(* Schneider Machine Expert - Basic project Proyecto_PLC_M221_Alex, file version 3.0.0.0 *)
(* CompanyInformations: Name=Alex, Country=España *)
(* ProjectInformations: Name=Proyecto1_PLC_M221_Alex, Description=Proyecto 1 Schneider Electric con M221.

Se ha a realizado el control de una maqueta Fischertechnik, la cual es una
línea de fabricación con dos máquinas herramienta, cinco cintas y dos selectores.

Se han realizado:
	- Diagrama de cableado de la maqueta.
	‐ Red de Petri
	‐ Implementación mediante Grafcet (las secciones LD)
	- Implementación de diferentes modos de la guía Gemma.
	‐ Implementar el panel de control de la máquina en un terminal de explotación. *)
(* UserInformations: LastName=Aquino Sala, FirstName=Alex, Email=aaleexsaalaa@gmail.com, Country=España *)

HARDWARE
  Cpu 0: TM221CE24R
  EthernetConfiguration: NetworkName=M221, IpAllocationMode=FixedAddress, IpAddress=10.7.1.158, SubnetMask=255.255.255.0
  SerialLineConfiguration: Baud=Baud19200, Parity=ParityEven, DataBits=DataBits8, StopBits=StopBits1, PhysicalMedium=PhysicalMediumRs485, TransmissionMode=TransmissionModeModbusRtu, SlaveId=1, Addressing=SlaveAddressing
  MastTask: UsePeriodScanMode=false, PeriodScan=100
  FastTask: Period=255
  CpuBehavior: StartingMode=StartAsPreviousState, AutoSaveRamOnEeprom=true, WatchdogPeriod=250

SYMBOLS  (address, symbol, comment, settings)
  %M100     AUTO  "Bit para poner el modo automatico"
  %M101     G_QCINTA1  "Bit para el control del modo manual"
  %M102     G_QCINTA2  "Bit para el control del modo manual"
  %M103     G_QCINTA3  "Bit para el control del modo manual"
  %M104     G_QCINTA4  "Bit para el control del modo manual"
  %M105     G_QMAC1  "Bit para el control del modo manual"
  %M106     G_QMAC2  "Bit para el control del modo manual"
  %M107     G_QSEL1AVANZA  "Bit para el control del modo manual"
  %M108     G_QSEL1RETRO  "Bit para el control del modo manual"
  %M109     G_QSEL2AVANZA  "Bit para el control del modo manual"
  %M110     G_QSEL2RETRO  "Bit para el control del modo manual"
  %M111     MARCHA
  %M112     EMERGENCIA  "Bit emergencia"
  %M113     REARME  "Bit de rearme"
  %M200     ESTOY_EMERG  "Bit que indica que esta en emergencia"
  %M201     ESTOY_MANUAL  "Bit para indicar cuando estamos en manual"
  %M202     ESTOY_AUTO  "Bit que indica cuando esta en modo automatico"
  %M300     PROBLEMAC1  "Problema en cinta 1"
  %M301     PROBLEMAC2  "Problema en cinta 2"
  %M302     PROBLEMAC3  "Problema en cinta 3"
  %M303     PROBLEMAC4  "Problema en cinta 4"
  %M304     PROBLEMA_MQ1  "Problema en maquina 1"
  %M305     PROBLEMA_MQ2  "Problema en maquina 2"
  %S9       SB_FALLBACKOUTPUT  "Establézcalo en 1 para aplicar retornos en salidas digitales y analógicas"
  %S23      SB_FREEZEGRAFCET  "Cuando es 1, valida el posicionamiento previo del GRAFCET. Si se mantiene este bit en 1, se inmoviliza el GRAFCET (se inmoviliza el gráfico)"
  %X2         "C1 avanza"
  %X3         "Espera C1"
  %X4         "R1 avanza"
  %X5         "C2 avanza"
  %X6         "Maquina 1 trabaja"
  %X8         "Maquina 2 trabaja"
  %X9         "Maquina 2 trabaja"
  %X10        "Espera M2"
  %X11        "C3 avanza"
  %X12        "R2 avanza"
  %X13        "C4 avanza"
  %X15        "R1 retrocede"
  %X16        "Espera"
  %X17        "R2 avanza"
  %X18        "Espera"
  %X19        "C1 avanza"
  %X20        "Epera R1"
  %X21        "Espera R2"
  %X23        "F4"
  %X24        "A6"
  %X25        "F1"
  %TM0        "Temporizador para los segundos de la maquina 1"  [Preset=5, Base=OneSecond]
  %TM1        "Temporizador para los segundos de la maquina 2"  [Preset=10, Base=OneSecond]
  %TM2        "Temporizador para que llegue la pieza al final de la cinta"  [Preset=7, Base=OneHundredMilliSeconds]
  %TM3        "Temporizador para que llegue la pieza al final de la cinta"  [Preset=2, Base=OneSecond]
  %TM4        "Temporizador que controla los problemas"  [Preset=7, Base=OneSecond]
  %TM5        "Temporizador que controla los problemas"  [Preset=7, Base=OneSecond]
  %TM6        "Temporizador que controla los problemas"  [Preset=7, Base=OneSecond]
  %TM7        "Temporizador que controla los problemas"  [Preset=7, Base=OneSecond]
  %TM8        "Temporizador que controla los problemas"  [Preset=7, Base=OneSecond]
  %TM9        "Temporizador que controla los problemas"  [Preset=12, Base=OneSecond]
  %I0.0     ISEL1FIN  "selector 1"
  %I0.1     ISENSORC1  "sensor 1"
  %I0.2     ISENSORCARGA
  %I0.3     ISENSORMAQ1  "sensor maquina"
  %I0.4     ISENSORMAQ2  "sensor maquina 2"
  %I0.5     ISEL1INI  "Selecrtor 1"
  %I0.6     ISENSORC4  "sensor 4"
  %I0.7     ISEL2FIN  "selecotr 2 fin"
  %I0.8     ISEL2INI  "Selector 2 ini"
  %Q0.0     QSEL1AVANZA  "Bit para mover el selector"
  %Q0.1     QMAQ1  "Bit para activar la maquina 1"
  %Q0.2     QCINTA3  "Bit para mover la cinta 3"
  %Q0.3     QSEL1RETRO  "Bit para mover el selector"
  %Q0.4     QSEL2AVANZA  "Bit para mover el selector"
  %Q0.5     QCINTA1  "Bit para mover la cinta 1"
  %Q0.6     QCINTA2  "Bit para mover la cinta 2"
  %Q0.7     QSEL2RETRO  "Bit para mover el selector"
  %Q0.8     QMAQ2  "Bit para activar la maquina"
  %Q0.9     QCINTA4  "Bit para mover la cinta 4"

GRAFCET GEMMA
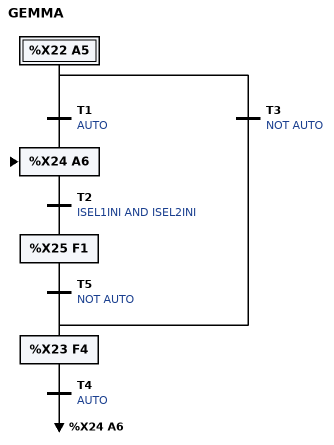
  INITIAL_STEP %X22  (* A5 *)
  STEP %X23  (* F4 *)
  STEP %X24  (* A6 *)
  STEP %X25  (* F1 *)
  TRANSITION T1 FROM %X22 TO %X24 := AUTO;
  TRANSITION T2 FROM %X24 TO %X25 := ISEL1INI AND ISEL2INI;
  TRANSITION T3 FROM %X22 TO %X23 := NOT AUTO;
  TRANSITION T4 FROM %X23 TO %X24 := AUTO;
  TRANSITION T5 FROM %X25 TO %X23 := NOT AUTO;

GRAFCET GRAFET
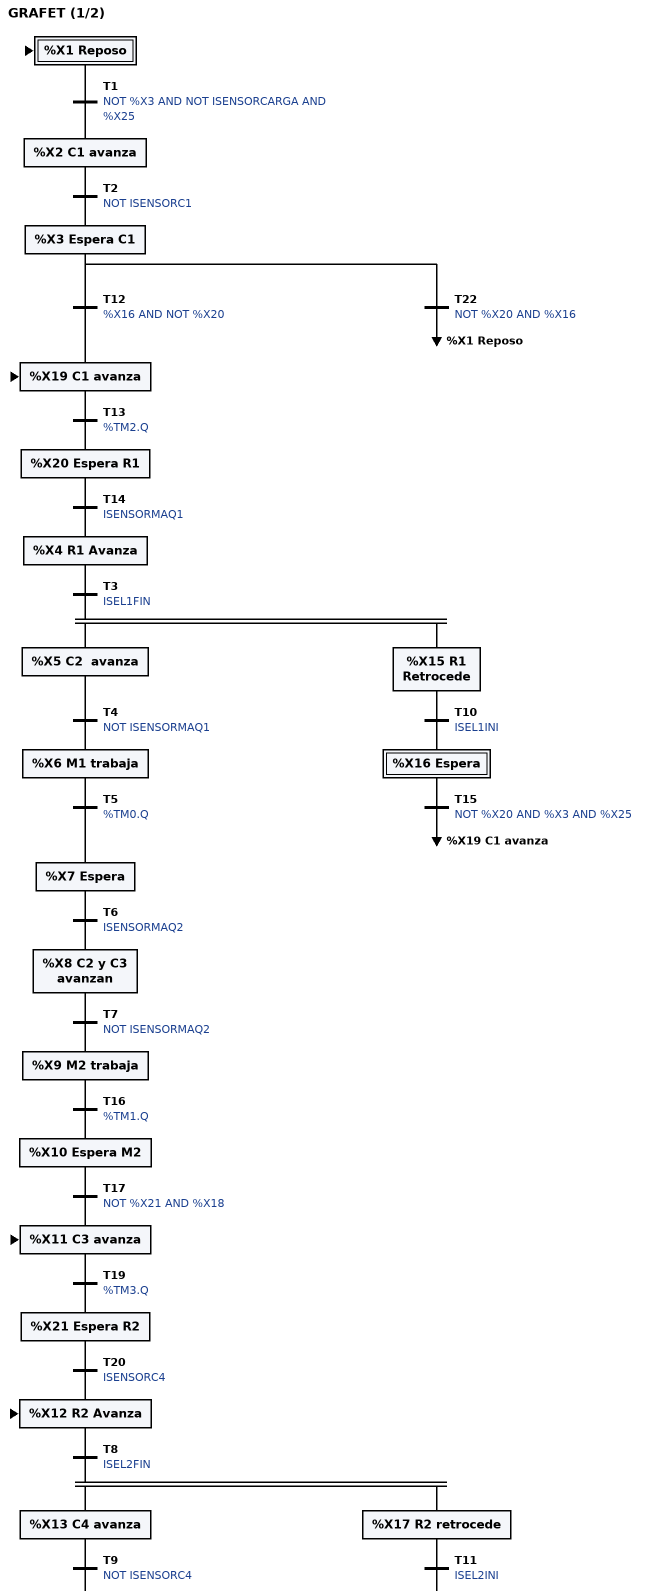
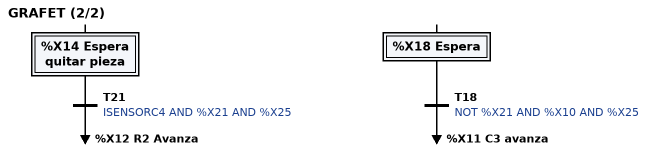
  INITIAL_STEP %X1  (* Reposo *)
  STEP %X2  (* C1 avanza *)
  STEP %X3  (* Espera C1 *)
  STEP %X4  (* R1 Avanza *)
  STEP %X5  (* C2  avanza *)
  STEP %X6  (* M1 trabaja *)
  STEP %X7  (* Espera *)
  STEP %X8  (* C2 y C3 avanzan *)
  STEP %X9  (* M2 trabaja *)
  STEP %X10  (* Espera M2 *)
  STEP %X11  (* C3 avanza *)
  STEP %X12  (* R2 Avanza *)
  STEP %X13  (* C4 avanza *)
  INITIAL_STEP %X14  (* Espera quitar pieza *)
  STEP %X15  (* R1 Retrocede *)
  INITIAL_STEP %X16  (* Espera  *)
  STEP %X17  (* R2 retrocede *)
  INITIAL_STEP %X18  (* Espera *)
  STEP %X19  (* C1 avanza *)
  STEP %X20  (* Espera R1 *)
  STEP %X21  (* Espera R2 *)
  TRANSITION T1 FROM %X1 TO %X2 := NOT %X3 AND NOT ISENSORCARGA AND %X25;
  TRANSITION T2 FROM %X2 TO %X3 := NOT ISENSORC1;
  TRANSITION T3 FROM %X4 TO %X5, %X15 := ISEL1FIN;
  TRANSITION T4 FROM %X5 TO %X6 := NOT ISENSORMAQ1;
  TRANSITION T5 FROM %X6 TO %X7 := %TM0.Q;
  TRANSITION T6 FROM %X7 TO %X8 := ISENSORMAQ2;
  TRANSITION T7 FROM %X8 TO %X9 := NOT ISENSORMAQ2;
  TRANSITION T8 FROM %X12 TO %X13, %X17 := ISEL2FIN;
  TRANSITION T9 FROM %X13 TO %X14 := NOT ISENSORC4;
  TRANSITION T10 FROM %X15 TO %X16 := ISEL1INI;
  TRANSITION T11 FROM %X17 TO %X18 := ISEL2INI;
  TRANSITION T12 FROM %X3 TO %X19 := %X16 AND NOT %X20;
  TRANSITION T13 FROM %X19 TO %X20 := %TM2.Q;
  TRANSITION T14 FROM %X20 TO %X4 := ISENSORMAQ1;
  TRANSITION T15 FROM %X16 TO %X19 := NOT %X20 AND %X3 AND %X25;
  TRANSITION T16 FROM %X9 TO %X10 := %TM1.Q;
  TRANSITION T17 FROM %X10 TO %X11 := NOT %X21 AND %X18;
  TRANSITION T18 FROM %X18 TO %X11 := NOT %X21 AND %X10 AND %X25;
  TRANSITION T19 FROM %X11 TO %X21 := %TM3.Q;
  TRANSITION T20 FROM %X21 TO %X12 := ISENSORC4;
  TRANSITION T21 FROM %X14 TO %X12 := ISENSORC4 AND %X21 AND %X25;
  TRANSITION T22 FROM %X3 TO %X1 := NOT %X20 AND %X16;

TRANSITION T1 (%X22 -> %X24) 
  (* SectionNumber=0 *)

// Rung 0: AUTO
  LD %M100                (* AUTO *)
  ENDT
  // as ST:
  //   TRANSITION := AUTO;

TRANSITION T2 (%X24 -> %X25) 
  (* SectionNumber=0 *)

// Rung 1: Tr2
  LD %I0.5                (* ISEL1INI *)
  AND %I0.8               (* ISEL2INI *)
  ENDT
  // as ST:
  //   TRANSITION := ISEL1INI AND ISEL2INI;

TRANSITION T3 (%X22 -> %X23) 
  (* SectionNumber=0 *)

// Rung 2: MANUAL
  LDN %M100               (* AUTO *)
  ENDT
  // as ST:
  //   TRANSITION := NOT AUTO;

TRANSITION T4 (%X23 -> %X24) 
  (* SectionNumber=0 *)

// Rung 3: AUTO
  LD %M100                (* AUTO *)
  ENDT
  // as ST:
  //   TRANSITION := AUTO;

TRANSITION T5 (%X25 -> %X23) 
  (* SectionNumber=0 *)

// Rung 4: MANUAL
  LDN %M100               (* AUTO *)
  ENDT
  // as ST:
  //   TRANSITION := NOT AUTO;

TRANSITION T1 (%X1 -> %X2) 
  (* SectionNumber=0 *)

// Rung 5: Tr1
  LDN %X3
  ANDN %I0.2              (* ISENSORCARGA *)
  AND %X25
  ENDT
  // as ST:
  //   TRANSITION := NOT %X3 AND NOT ISENSORCARGA AND %X25;

TRANSITION T2 (%X2 -> %X3) 
  (* SectionNumber=0 *)

// Rung 6: Tr2
  LDN %I0.1               (* ISENSORC1 *)
  ENDT
  // as ST:
  //   TRANSITION := NOT ISENSORC1;

TRANSITION T3 (%X4 -> %X5, %X15) 
  (* SectionNumber=0 *)

// Rung 7: Tr4
  LD %I0.0                (* ISEL1FIN *)
  ENDT
  // as ST:
  //   TRANSITION := ISEL1FIN;

TRANSITION T4 (%X5 -> %X6) 
  (* SectionNumber=0 *)

// Rung 8: Tr5
  LDN %I0.3               (* ISENSORMAQ1 *)
  ENDT
  // as ST:
  //   TRANSITION := NOT ISENSORMAQ1;

TRANSITION T5 (%X6 -> %X7) 
  (* SectionNumber=0 *)

// Rung 9: Temp
  LD %TM0.Q
  ENDT
  // as ST:
  //   TRANSITION := %TM0.Q;

TRANSITION T6 (%X7 -> %X8) 
  (* SectionNumber=0 *)

// Rung 10: Tr7
  LD %I0.4                (* ISENSORMAQ2 *)
  ENDT
  // as ST:
  //   TRANSITION := ISENSORMAQ2;

TRANSITION T7 (%X8 -> %X9) 
  (* SectionNumber=0 *)

// Rung 11: Tr8
  LDN %I0.4               (* ISENSORMAQ2 *)
  ENDT
  // as ST:
  //   TRANSITION := NOT ISENSORMAQ2;

TRANSITION T8 (%X12 -> %X13, %X17) 
  (* SectionNumber=0 *)

// Rung 12: Tr12
  LD %I0.7                (* ISEL2FIN *)
  ENDT
  // as ST:
  //   TRANSITION := ISEL2FIN;

TRANSITION T9 (%X13 -> %X14) 
  (* SectionNumber=0 *)

// Rung 13: Tr13
  LDN %I0.6               (* ISENSORC4 *)
  ENDT
  // as ST:
  //   TRANSITION := NOT ISENSORC4;

TRANSITION T10 (%X15 -> %X16) 
  (* SectionNumber=0 *)

// Rung 14: Tr14
  LD %I0.5                (* ISEL1INI *)
  ENDT
  // as ST:
  //   TRANSITION := ISEL1INI;

TRANSITION T11 (%X17 -> %X18) 
  (* SectionNumber=0 *)

// Rung 15: Tr16
  LD %I0.8                (* ISEL2INI *)
  ENDT
  // as ST:
  //   TRANSITION := ISEL2INI;

TRANSITION T12 (%X3 -> %X19) 
  (* SectionNumber=0 *)

// Rung 16: Tr3
  LD %X16
  ANDN %X20
  ENDT
  // as ST:
  //   TRANSITION := %X16 AND NOT %X20;

TRANSITION T13 (%X19 -> %X20) 
  (* SectionNumber=0 *)

// Rung 17: Temp
  LD %TM2.Q
  ENDT
  // as ST:
  //   TRANSITION := %TM2.Q;

TRANSITION T14 (%X20 -> %X4) 
  (* SectionNumber=0 *)

// Rung 18: Tr19
  LD %I0.3                (* ISENSORMAQ1 *)
  ENDT
  // as ST:
  //   TRANSITION := ISENSORMAQ1;

TRANSITION T15 (%X16 -> %X19) 
  (* SectionNumber=0 *)

// Rung 19: Tr20
  LDN %X20
  AND %X3
  AND %X25
  ENDT
  // as ST:
  //   TRANSITION := NOT %X20 AND %X3 AND %X25;

TRANSITION T16 (%X9 -> %X10) 
  (* SectionNumber=0 *)

// Rung 20: Temp
  LD %TM1.Q
  ENDT
  // as ST:
  //   TRANSITION := %TM1.Q;

TRANSITION T17 (%X10 -> %X11) 
  (* SectionNumber=0 *)

// Rung 21: Tr13
  LDN %X21
  AND %X18
  ENDT
  // as ST:
  //   TRANSITION := NOT %X21 AND %X18;

TRANSITION T18 (%X18 -> %X11) 
  (* SectionNumber=0 *)

// Rung 22: Tr13
  LDN %X21
  AND %X10
  AND %X25
  ENDT
  // as ST:
  //   TRANSITION := NOT %X21 AND %X10 AND %X25;

TRANSITION T19 (%X11 -> %X21) 
  (* SectionNumber=0 *)

// Rung 23: Temp
  LD %TM3.Q
  ENDT
  // as ST:
  //   TRANSITION := %TM3.Q;

TRANSITION T20 (%X21 -> %X12) 
  (* SectionNumber=0 *)

// Rung 24: Tr14
  LD %I0.6                (* ISENSORC4 *)
  ENDT
  // as ST:
  //   TRANSITION := ISENSORC4;

TRANSITION T21 (%X14 -> %X12) 
  (* SectionNumber=0 *)

// Rung 25: Tr21
  LD %I0.6                (* ISENSORC4 *)
  AND %X21
  AND %X25
  ENDT
  // as ST:
  //   TRANSITION := ISENSORC4 AND %X21 AND %X25;

TRANSITION T22 (%X3 -> %X1) 
  (* SectionNumber=0 *)

// Rung 26: Tr22
  LDN %X20
  AND %X16
  ENDT
  // as ST:
  //   TRANSITION := NOT %X20 AND %X16;

POU SALIDAS  (* Lineas para controlar las salidas de nuestro sistema *)
  (* SectionNumber=27 *)

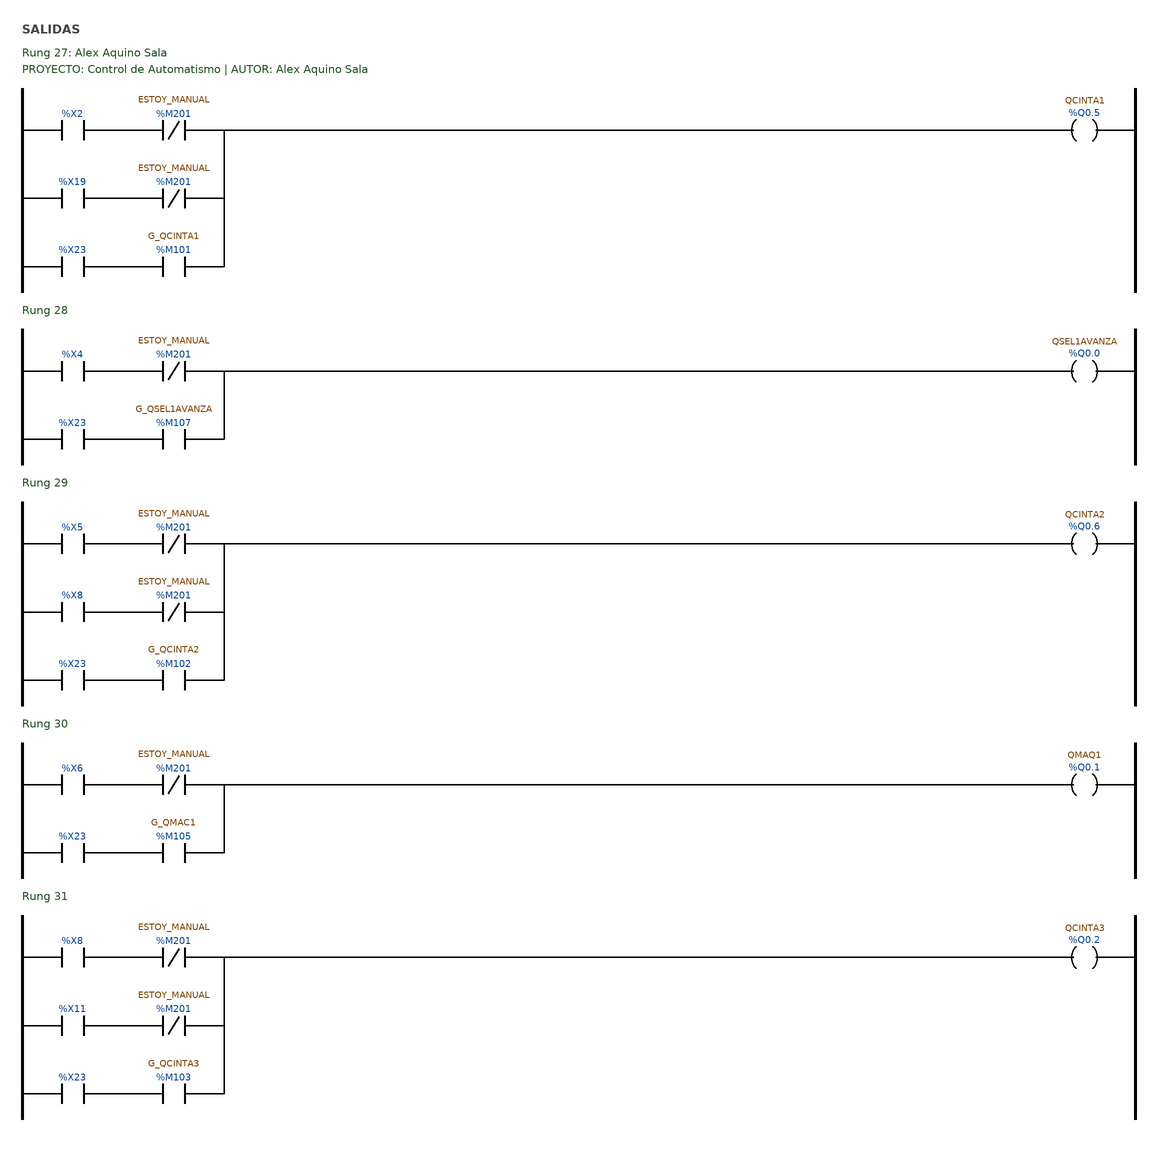

// Rung 27: Alex Aquino Sala
// PROYECTO: Control de Automatismo | AUTOR: Alex Aquino Sala
  LD %X2
  ANDN %M201              (* ESTOY_MANUAL *)
  OR( %X19
  ANDN %M201              (* ESTOY_MANUAL *)
  )
  OR( %X23
  AND %M101               (* G_QCINTA1 *)
  )
  ST %Q0.5                (* QCINTA1 *)
  // as ST:
  //   QCINTA1 := %X2 AND NOT ESTOY_MANUAL OR %X19 AND NOT ESTOY_MANUAL OR %X23 AND G_QCINTA1;

// Rung 28
  LD %X4
  ANDN %M201              (* ESTOY_MANUAL *)
  OR( %X23
  AND %M107               (* G_QSEL1AVANZA *)
  )
  ST %Q0.0                (* QSEL1AVANZA *)
  // as ST:
  //   QSEL1AVANZA := %X4 AND NOT ESTOY_MANUAL OR %X23 AND G_QSEL1AVANZA;

// Rung 29
  LD %X5
  ANDN %M201              (* ESTOY_MANUAL *)
  OR( %X8
  ANDN %M201              (* ESTOY_MANUAL *)
  )
  OR( %X23
  AND %M102               (* G_QCINTA2 *)
  )
  ST %Q0.6                (* QCINTA2 *)
  // as ST:
  //   QCINTA2 := %X5 AND NOT ESTOY_MANUAL OR %X8 AND NOT ESTOY_MANUAL OR %X23 AND G_QCINTA2;

// Rung 30
  LD %X6
  ANDN %M201              (* ESTOY_MANUAL *)
  OR( %X23
  AND %M105               (* G_QMAC1 *)
  )
  ST %Q0.1                (* QMAQ1 *)
  // as ST:
  //   QMAQ1 := %X6 AND NOT ESTOY_MANUAL OR %X23 AND G_QMAC1;

// Rung 31
  LD %X8
  ANDN %M201              (* ESTOY_MANUAL *)
  OR( %X11
  ANDN %M201              (* ESTOY_MANUAL *)
  )
  OR( %X23
  AND %M103               (* G_QCINTA3 *)
  )
  ST %Q0.2                (* QCINTA3 *)
  // as ST:
  //   QCINTA3 := %X8 AND NOT ESTOY_MANUAL OR %X11 AND NOT ESTOY_MANUAL OR %X23 AND G_QCINTA3;

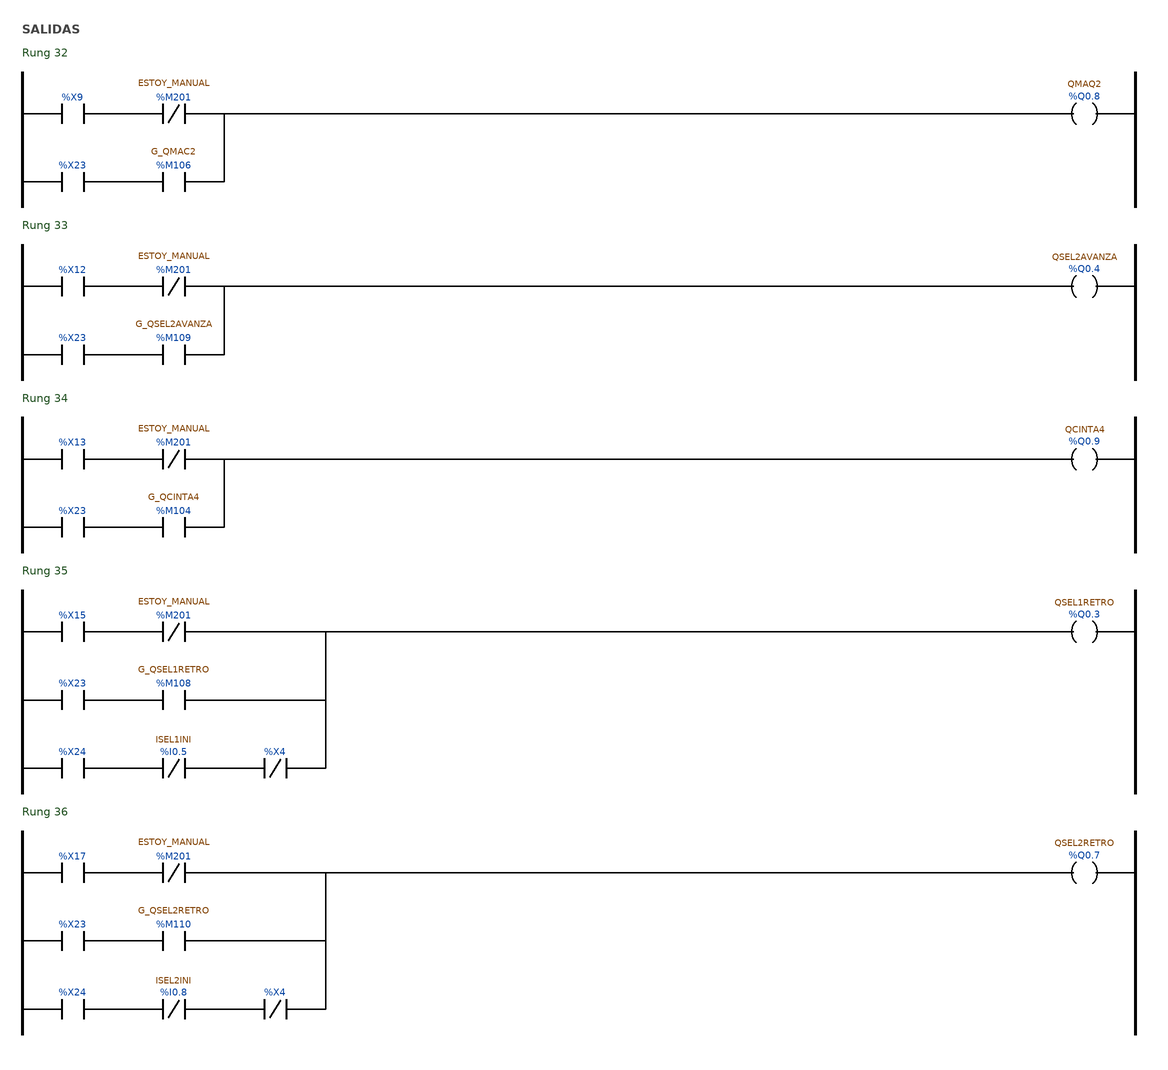

// Rung 32
  LD %X9
  ANDN %M201              (* ESTOY_MANUAL *)
  OR( %X23
  AND %M106               (* G_QMAC2 *)
  )
  ST %Q0.8                (* QMAQ2 *)
  // as ST:
  //   QMAQ2 := %X9 AND NOT ESTOY_MANUAL OR %X23 AND G_QMAC2;

// Rung 33
  LD %X12
  ANDN %M201              (* ESTOY_MANUAL *)
  OR( %X23
  AND %M109               (* G_QSEL2AVANZA *)
  )
  ST %Q0.4                (* QSEL2AVANZA *)
  // as ST:
  //   QSEL2AVANZA := %X12 AND NOT ESTOY_MANUAL OR %X23 AND G_QSEL2AVANZA;

// Rung 34
  LD %X13
  ANDN %M201              (* ESTOY_MANUAL *)
  OR( %X23
  AND %M104               (* G_QCINTA4 *)
  )
  ST %Q0.9                (* QCINTA4 *)
  // as ST:
  //   QCINTA4 := %X13 AND NOT ESTOY_MANUAL OR %X23 AND G_QCINTA4;

// Rung 35
  LD %X15
  ANDN %M201              (* ESTOY_MANUAL *)
  OR( %X23
  AND %M108               (* G_QSEL1RETRO *)
  )
  OR( %X24
  ANDN %I0.5              (* ISEL1INI *)
  ANDN %X4
  )
  ST %Q0.3                (* QSEL1RETRO *)
  // as ST:
  //   QSEL1RETRO := %X15 AND NOT ESTOY_MANUAL OR %X23 AND G_QSEL1RETRO OR %X24 AND NOT ISEL1INI AND NOT %X4;

// Rung 36
  LD %X17
  ANDN %M201              (* ESTOY_MANUAL *)
  OR( %X23
  AND %M110               (* G_QSEL2RETRO *)
  )
  OR( %X24
  ANDN %I0.8              (* ISEL2INI *)
  ANDN %X4
  )
  ST %Q0.7                (* QSEL2RETRO *)
  // as ST:
  //   QSEL2RETRO := %X17 AND NOT ESTOY_MANUAL OR %X23 AND G_QSEL2RETRO OR %X24 AND NOT ISEL2INI AND NOT %X4;

POU MODOS  (* Lineas para comunicar con el HMI *)
  (* SectionNumber=28 *)

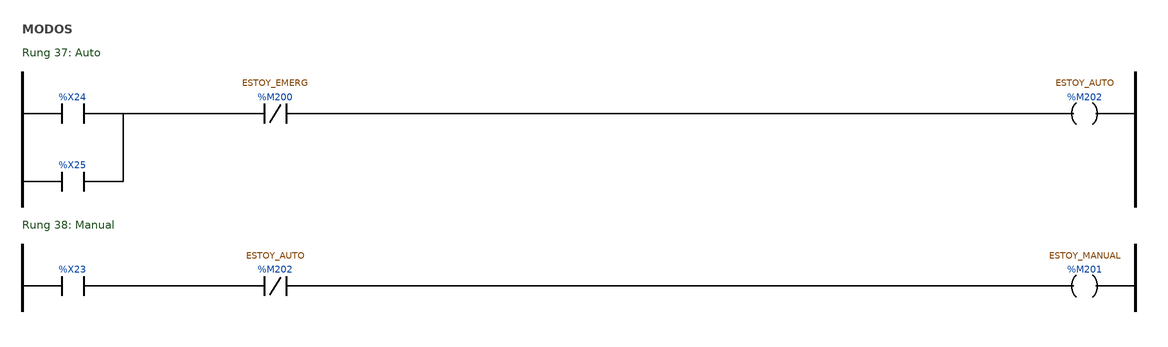

// Rung 37: Auto
  LD %X24
  OR %X25
  ANDN %M200              (* ESTOY_EMERG *)
  ST %M202                (* ESTOY_AUTO *)
  // as ST:
  //   ESTOY_AUTO := (%X24 OR %X25) AND NOT ESTOY_EMERG;

// Rung 38: Manual
  LD %X23
  ANDN %M202              (* ESTOY_AUTO *)
  ST %M201                (* ESTOY_MANUAL *)
  // as ST:
  //   ESTOY_MANUAL := %X23 AND NOT ESTOY_AUTO;

POU TEMPORIZADORES
  (* SectionNumber=29 *)

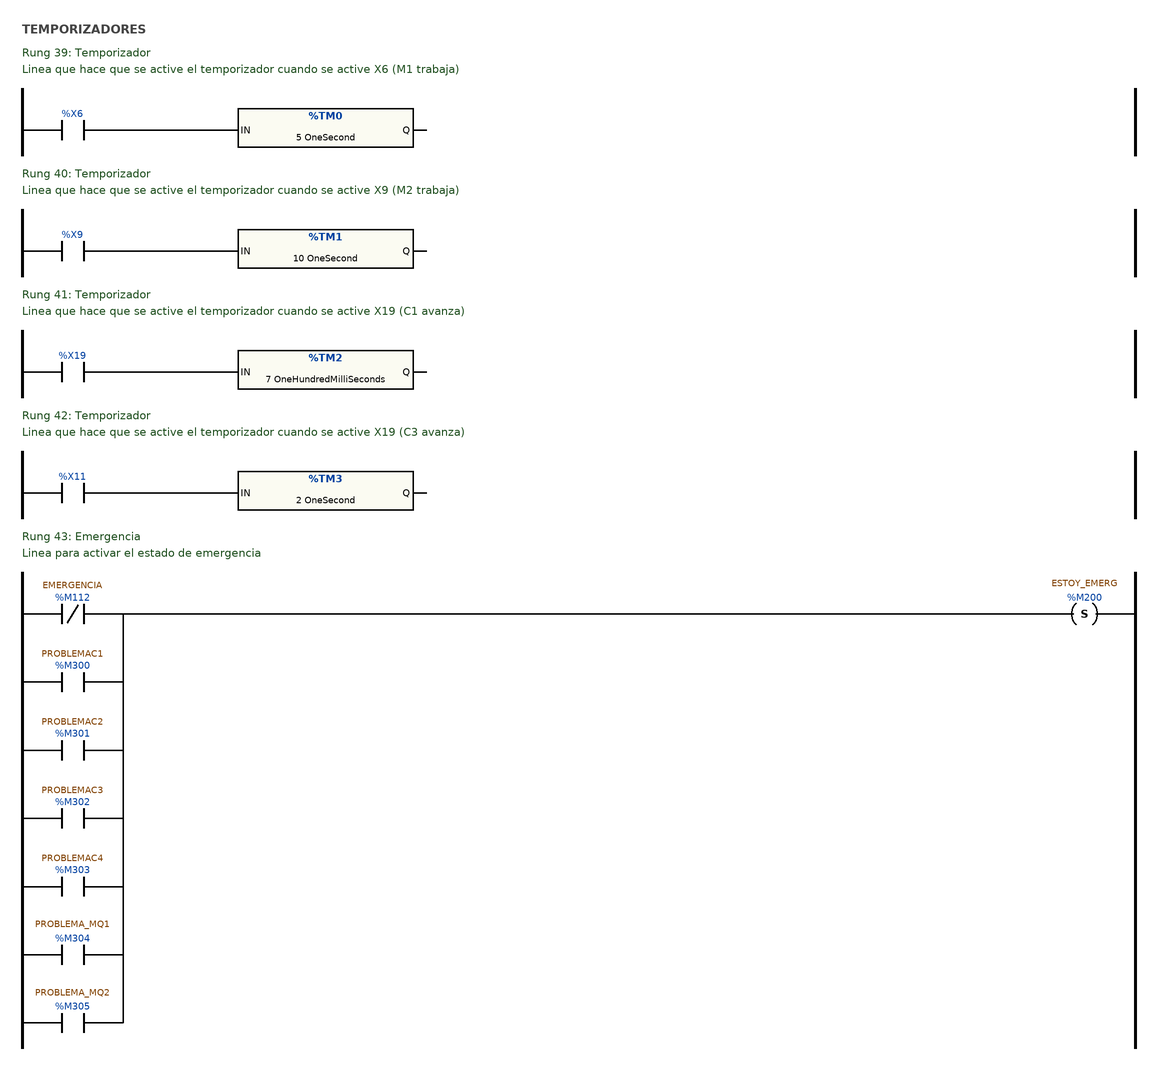

// Rung 39: Temporizador
// Linea que hace que se active el temporizador cuando se active X6 (M1 trabaja)
  BLK %TM0
  LD %X6
  IN
  END_BLK
  // as ST:
  //   %TM0(IN := %X6);

// Rung 40: Temporizador
// Linea que hace que se active el temporizador cuando se active X9 (M2 trabaja)
  BLK %TM1
  LD %X9
  IN
  END_BLK
  // as ST:
  //   %TM1(IN := %X9);

// Rung 41: Temporizador
// Linea que hace que se active el temporizador cuando se active X19 (C1 avanza)
  BLK %TM2
  LD %X19
  IN
  END_BLK
  // as ST:
  //   %TM2(IN := %X19);

// Rung 42: Temporizador
// Linea que hace que se active el temporizador cuando se active X19 (C3 avanza)
  BLK %TM3
  LD %X11
  IN
  END_BLK
  // as ST:
  //   %TM3(IN := %X11);

// Rung 43: Emergencia
// Linea para activar el estado de emergencia
  LDN %M112               (* EMERGENCIA *)
  OR %M300                (* PROBLEMAC1 *)
  OR %M301                (* PROBLEMAC2 *)
  OR %M302                (* PROBLEMAC3 *)
  OR %M303                (* PROBLEMAC4 *)
  OR %M304                (* PROBLEMA_MQ1 *)
  OR %M305                (* PROBLEMA_MQ2 *)
  S %M200                 (* ESTOY_EMERG *)
  // as ST:
  //   IF NOT EMERGENCIA OR PROBLEMAC1 OR PROBLEMAC2 OR PROBLEMAC3 OR PROBLEMAC4 OR PROBLEMA_MQ1 OR PROBLEMA_MQ2 THEN ESTOY_EMERG := TRUE; END_IF;

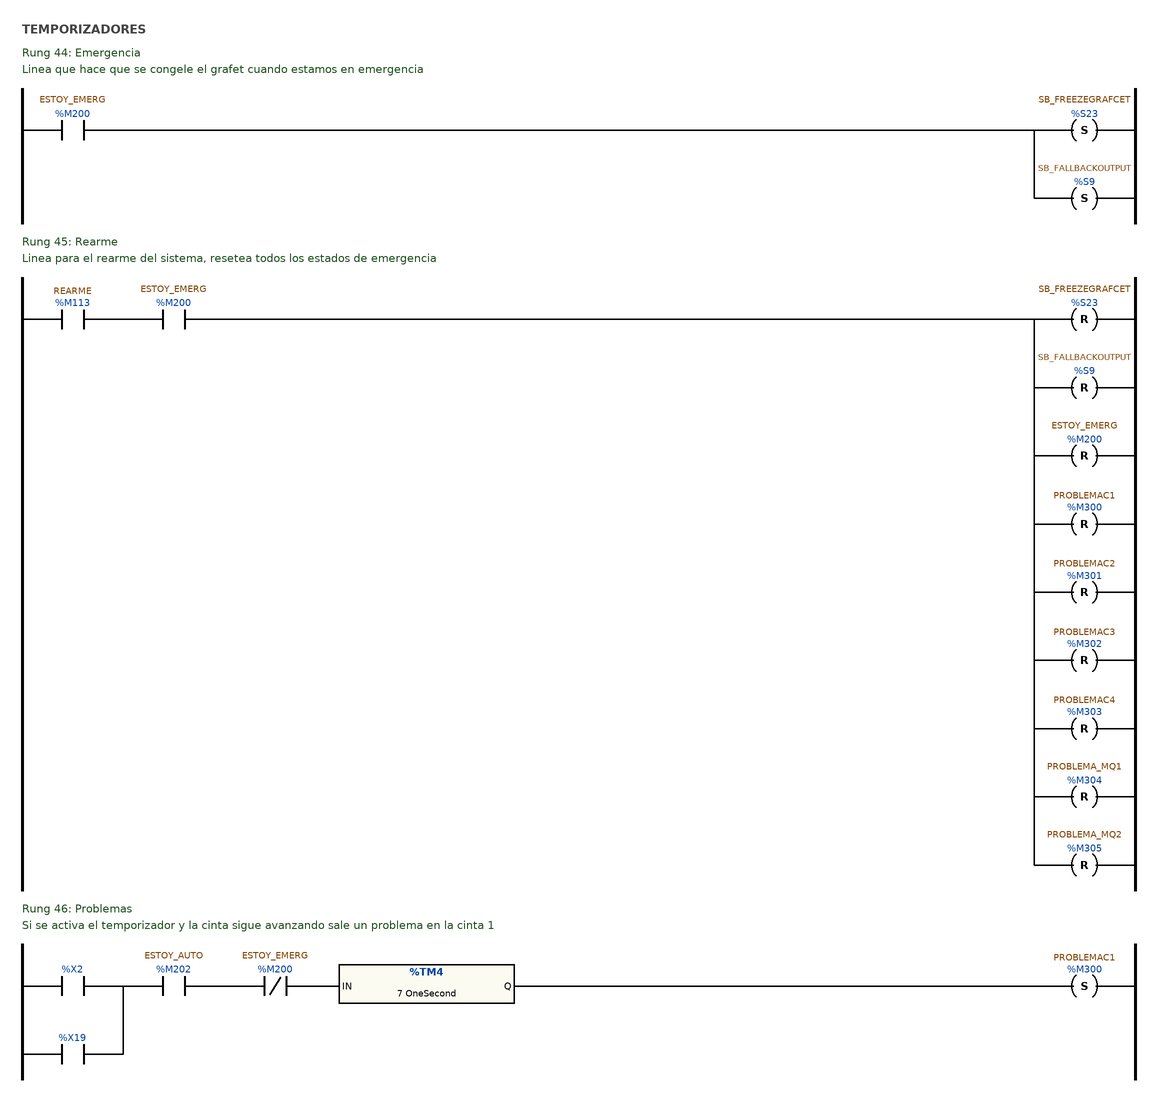

// Rung 44: Emergencia
// Linea que hace que se congele el grafet cuando estamos en emergencia
  LD %M200                (* ESTOY_EMERG *)
  S %S23                  (* SB_FREEZEGRAFCET *)
  S %S9                   (* SB_FALLBACKOUTPUT *)
  // as ST:
  //   IF ESTOY_EMERG THEN SB_FREEZEGRAFCET := TRUE; END_IF;
  //   IF ESTOY_EMERG THEN SB_FALLBACKOUTPUT := TRUE; END_IF;

// Rung 45: Rearme
// Linea para el rearme del sistema, resetea todos los estados de emergencia
  LD %M113                (* REARME *)
  AND %M200               (* ESTOY_EMERG *)
  R %S23                  (* SB_FREEZEGRAFCET *)
  R %S9                   (* SB_FALLBACKOUTPUT *)
  R %M200                 (* ESTOY_EMERG *)
  R %M300                 (* PROBLEMAC1 *)
  R %M301                 (* PROBLEMAC2 *)
  R %M302                 (* PROBLEMAC3 *)
  R %M303                 (* PROBLEMAC4 *)
  R %M304                 (* PROBLEMA_MQ1 *)
  R %M305                 (* PROBLEMA_MQ2 *)
  // as ST:
  //   IF REARME AND ESTOY_EMERG THEN SB_FREEZEGRAFCET := FALSE; END_IF;
  //   IF REARME AND ESTOY_EMERG THEN SB_FALLBACKOUTPUT := FALSE; END_IF;
  //   _t1 := REARME AND ESTOY_EMERG;
  //   IF _t1 THEN ESTOY_EMERG := FALSE; END_IF;
  //   IF _t1 THEN PROBLEMAC1 := FALSE; END_IF;
  //   IF _t1 THEN PROBLEMAC2 := FALSE; END_IF;
  //   IF _t1 THEN PROBLEMAC3 := FALSE; END_IF;
  //   IF _t1 THEN PROBLEMAC4 := FALSE; END_IF;
  //   IF _t1 THEN PROBLEMA_MQ1 := FALSE; END_IF;
  //   IF _t1 THEN PROBLEMA_MQ2 := FALSE; END_IF;

// Rung 46: Problemas
// Si se activa el temporizador y la cinta sigue avanzando sale un problema en la cinta 1
  BLK %TM4
  LD %X2
  OR %X19
  AND %M202               (* ESTOY_AUTO *)
  ANDN %M200              (* ESTOY_EMERG *)
  IN
  OUT_BLK
  LD Q
  S %M300                 (* PROBLEMAC1 *)
  END_BLK
  // as ST:
  //   %TM4(IN := (%X2 OR %X19) AND ESTOY_AUTO AND NOT ESTOY_EMERG);
  //   IF %TM4.Q THEN PROBLEMAC1 := TRUE; END_IF;

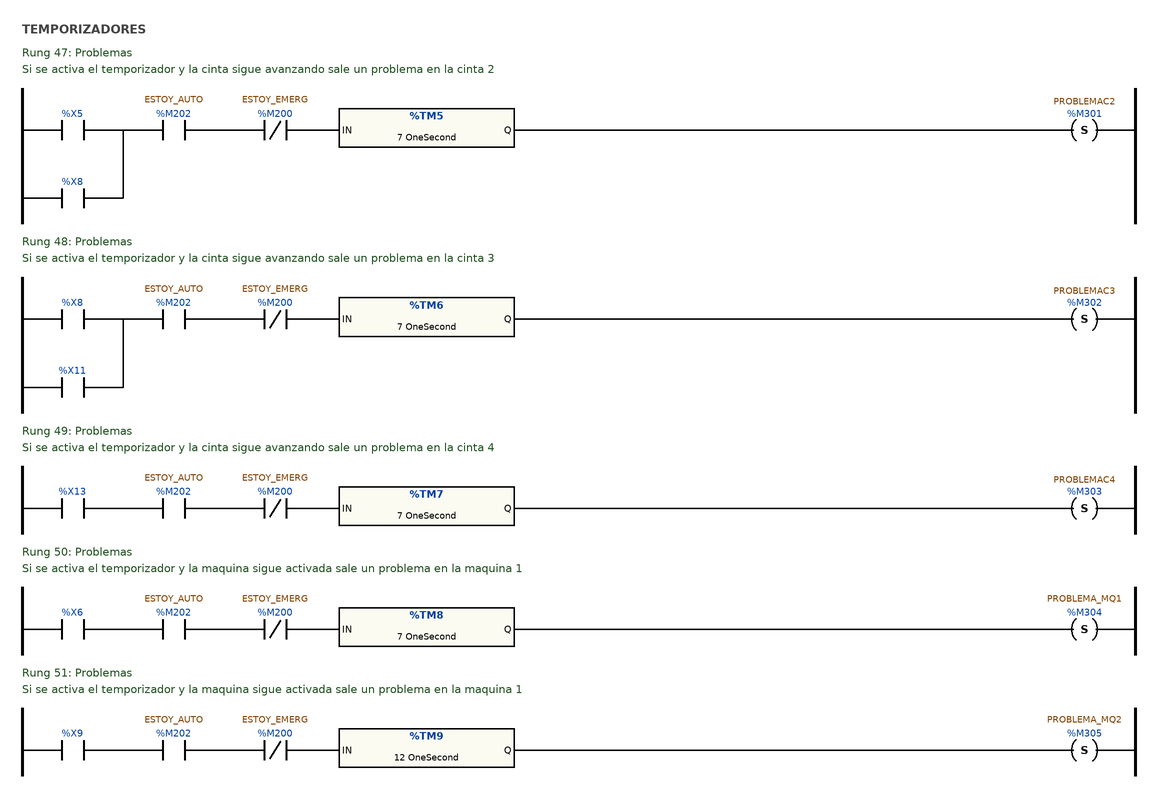

// Rung 47: Problemas
// Si se activa el temporizador y la cinta sigue avanzando sale un problema en la cinta 2
  BLK %TM5
  LD %X5
  OR %X8
  AND %M202               (* ESTOY_AUTO *)
  ANDN %M200              (* ESTOY_EMERG *)
  IN
  OUT_BLK
  LD Q
  S %M301                 (* PROBLEMAC2 *)
  END_BLK
  // as ST:
  //   %TM5(IN := (%X5 OR %X8) AND ESTOY_AUTO AND NOT ESTOY_EMERG);
  //   IF %TM5.Q THEN PROBLEMAC2 := TRUE; END_IF;

// Rung 48: Problemas
// Si se activa el temporizador y la cinta sigue avanzando sale un problema en la cinta 3
  BLK %TM6
  LD %X8
  OR %X11
  AND %M202               (* ESTOY_AUTO *)
  ANDN %M200              (* ESTOY_EMERG *)
  IN
  OUT_BLK
  LD Q
  S %M302                 (* PROBLEMAC3 *)
  END_BLK
  // as ST:
  //   %TM6(IN := (%X8 OR %X11) AND ESTOY_AUTO AND NOT ESTOY_EMERG);
  //   IF %TM6.Q THEN PROBLEMAC3 := TRUE; END_IF;

// Rung 49: Problemas
// Si se activa el temporizador y la cinta sigue avanzando sale un problema en la cinta 4
  BLK %TM7
  LD %X13
  AND %M202               (* ESTOY_AUTO *)
  ANDN %M200              (* ESTOY_EMERG *)
  IN
  OUT_BLK
  LD Q
  S %M303                 (* PROBLEMAC4 *)
  END_BLK
  // as ST:
  //   %TM7(IN := %X13 AND ESTOY_AUTO AND NOT ESTOY_EMERG);
  //   IF %TM7.Q THEN PROBLEMAC4 := TRUE; END_IF;

// Rung 50: Problemas
// Si se activa el temporizador y la maquina sigue activada sale un problema en la maquina 1
  BLK %TM8
  LD %X6
  AND %M202               (* ESTOY_AUTO *)
  ANDN %M200              (* ESTOY_EMERG *)
  IN
  OUT_BLK
  LD Q
  S %M304                 (* PROBLEMA_MQ1 *)
  END_BLK
  // as ST:
  //   %TM8(IN := %X6 AND ESTOY_AUTO AND NOT ESTOY_EMERG);
  //   IF %TM8.Q THEN PROBLEMA_MQ1 := TRUE; END_IF;

// Rung 51: Problemas
// Si se activa el temporizador y la maquina sigue activada sale un problema en la maquina 1
  BLK %TM9
  LD %X9
  AND %M202               (* ESTOY_AUTO *)
  ANDN %M200              (* ESTOY_EMERG *)
  IN
  OUT_BLK
  LD Q
  S %M305                 (* PROBLEMA_MQ2 *)
  END_BLK
  // as ST:
  //   %TM9(IN := %X9 AND ESTOY_AUTO AND NOT ESTOY_EMERG);
  //   IF %TM9.Q THEN PROBLEMA_MQ2 := TRUE; END_IF;
